Fanuc KAREL source: test_tpe.kl

PROGRAM test_tpe
%NOLOCKGROUP

%INCLUDE tpe.klh
%INCLUDE kunit.klh


BEGIN
END test_tpe
